// TwinCAT 3 PLC project Oefeningen4
// ProgramVersion: 3.1.4026.18
// libraries:
//   Tc2_BABasic, * (Beckhoff Automation GmbH)
//   Tc2_Standard, * (Beckhoff Automation GmbH)
//   Tc2_System, * (Beckhoff Automation GmbH)
//   Tc2_Utilities, * (Beckhoff Automation GmbH)
//   Tc3_Module, * (Beckhoff Automation GmbH)
// project tree:
//   DUTs/ DUT_Kamer.TcDUT
//   / GlobalTextList.TcGTLO, PlcTask.TcTTO, Visualization Manager.TcVMO (not stored)
//   POUs/ MAIN.TcPOU, MEAN.TcPOU, prg_Finale.TcPOU, prg_KantoorVerlichting.TcPOU, prg_Thermostaatregeling.TcPOU, prg_ThermostaatregelingTijdsturing.TcPOU
//   VISUs/ Visualization_Thermostaatregeling.TcVIS, Visualization_ThermostaatTijdsturing.TcVIS
// (motion and I/O tree: see PLC project oefeningen1)
// real-time tasks:
//   TASK PlcTask: cycle T#10ms, priority 20, ADS port 350
//   TASK PlcTask1: cycle T#10ms, priority 21, ADS port 351
//   TASK PlcTask2: cycle T#10ms, priority 22, ADS port 352
//   TASK PlcTask3: cycle T#10ms, priority 23, ADS port 353
//   TASK PlcTask4: cycle T#10ms, priority 24, ADS port 354

CONFIGURATION Oefeningen4
    RESOURCE PLC ON TwinCAT3
        TASK PlcTask(INTERVAL := T#10ms, PRIORITY := 23);
        PROGRAM MAIN WITH PlcTask : MAIN;
    END_RESOURCE
END_CONFIGURATION

// ---- DUTs/DUT_Kamer.TcDUT
TYPE DUT_Kamer :
STRUCT
    Licht : BOOL;
    Temperatuur : REAL;
    MA_Temp : REAL;
END_STRUCT
END_TYPE

// ---- POUs/MAIN.TcPOU
PROGRAM MAIN
VAR
END_VAR

//prg_KantoorVerlichting();
//prg_Thermostaatregeling();
prg_ThermostaatregelingTijdsturing();

END_PROGRAM

// ---- POUs/prg_ThermostaatregelingTijdsturing.TcPOU
PROGRAM prg_ThermostaatregelingTijdsturing
VAR
   	Temperatuur : REAL;            
    TempLog     : ARRAY[0..19] OF REAL;
    TempAlarm   : ARRAY[0..19] OF BOOL;
    idx         : INT := 0;        
    tSample     : TON;
END_VAR

// timer 1 seconde
tSample(IN := TRUE, PT := T#1S);
tSample();

IF tSample.Q THEN
    TempLog[idx] := Temperatuur;               // log huidige temperatuur
    TempAlarm[idx] := (Temperatuur < 10.0);   // alarm als <10°C
    idx := (idx + 1) MOD 20;                  // circular buffer
    tSample(IN := FALSE);
    tSample(IN := TRUE);
END_IF

END_PROGRAM

// ---- POUs/MEAN.TcPOU
FUNCTION MEAN : REAL
VAR_INPUT
    arr : ARRAY[1..10] OF REAL;
END_VAR

VAR
    i : INT;
    sum : REAL := 0.0;
END_VAR

FOR i := 1 TO 10 DO
    sum := sum + arr[i];
END_FOR

MEAN := sum / 10.0;

END_FUNCTION

// ---- POUs/prg_Finale.TcPOU
PROGRAM prg_Finale
VAR
    (* ---- Kamers ---- *)
    Woonkamer : DUT_Kamer := (Temperatuur := 21.0);
    Keuken    : DUT_Kamer := (Temperatuur := 20.5);
    Badkamer  : DUT_Kamer := (Temperatuur := 22.0);
    Gang      : DUT_Kamer := (Temperatuur := 19.5);

    (* ---- 10s timer ---- *)
    tMeasure : TON;

    (* ---- Moving Average buffers (10 waarden) ---- *)
    TempBuf_WK : ARRAY[1..10] OF REAL;
    TempBuf_K  : ARRAY[1..10] OF REAL;
    TempBuf_B  : ARRAY[1..10] OF REAL;
    TempBuf_G  : ARRAY[1..10] OF REAL;

    idx : INT := 1; (* circulaire index 1..10 *)

    (* ---- Logging MA + timestamp (laatste 20 waarden) ---- *)
    LogMA : ARRAY[1..20, 1..2] OF LREAL;
    (* Kolom 1 = timestamp (s), Kolom 2 = MA temperatuur *)

    logIndex : INT := 1;

    sysTime : LTIME;

    (* ---- VISU toggles ---- *)
    VISU_Toggle_WK : BOOL;
    VISU_Toggle_K  : BOOL;
    VISU_Toggle_B  : BOOL;
    VISU_Toggle_G  : BOOL;

    VISU_ShowTemp : BOOL;
END_VAR

(* Start 10s timer *)
tMeasure(IN := TRUE, PT := T#10s);

(* ---- Licht toggles (via visualisatie) ---- *)
IF VISU_Toggle_WK THEN
    Woonkamer.Licht := NOT Woonkamer.Licht;
    VISU_Toggle_WK := FALSE;
END_IF

IF VISU_Toggle_K THEN
    Keuken.Licht := NOT Keuken.Licht;
    VISU_Toggle_K := FALSE;
END_IF

IF VISU_Toggle_B THEN
    Badkamer.Licht := NOT Badkamer.Licht;
    VISU_Toggle_B := FALSE;
END_IF

IF VISU_Toggle_G THEN
    Gang.Licht := NOT Gang.Licht;
    VISU_Toggle_G := FALSE;
END_IF

(* ---- Elke 10 seconden meten ---- *)
IF tMeasure.Q THEN

    (* Simuleer temperatuur (later vervang je dit door echte sensor) *)
    Woonkamer.Temperatuur := Woonkamer.Temperatuur + (RAND() - 0.5) * 0.2;
    Keuken.Temperatuur    := Keuken.Temperatuur + (RAND() - 0.5) * 0.2;
    Badkamer.Temperatuur  := Badkamer.Temperatuur + (RAND() - 0.5) * 0.2;
    Gang.Temperatuur      := Gang.Temperatuur + (RAND() - 0.5) * 0.2;

    (* ---- Circulaire buffer update ---- *)
    idx := idx + 1;
    IF idx > 10 THEN
        idx := 1;
    END_IF

    TempBuf_WK[idx] := Woonkamer.Temperatuur;
    TempBuf_K[idx]  := Keuken.Temperatuur;
    TempBuf_B[idx]  := Badkamer.Temperatuur;
    TempBuf_G[idx]  := Gang.Temperatuur;

    (* ---- Bereken Moving Average ---- *)
    Woonkamer.MA_Temp := MEAN(TempBuf_WK);
    Keuken.MA_Temp    := MEAN(TempBuf_K);
    Badkamer.MA_Temp  := MEAN(TempBuf_B);
    Gang.MA_Temp      := MEAN(TempBuf_G);

    (* ---- Timestamp ---- *)
    sysTime := F_GetCurTime();

    (* ---- Log laatste 20 MA waarden (voor tabel in VISU) ---- *)
    LogMA[logIndex,1] := LTIME_TO_LREAL(sysTime) / 1_000_000_000.0; (* seconden *)
    LogMA[logIndex,2] := Woonkamer.MA_Temp; (* je kan hier ook andere kamer kiezen *)

    logIndex := logIndex + 1;
    IF logIndex > 20 THEN
        logIndex := 1;
    END_IF

    (* Reset timer *)
    tMeasure(IN := FALSE);
END_IF

END_PROGRAM

// ---- POUs/prg_KantoorVerlichting.TcPOU
PROGRAM prg_KantoorVerlichting
VAR
	bSchakelaar_1		AT		%I*		:BOOL;
	bSchakelaar_2		AT		%I*		:BOOL;
	bSchakelaar_3		AT		%I*		:BOOL;
	bVerlichting	 	AT 		%Q* 	:BOOL;

	LichtVerlengen: TON;
	TimerVerlichting: TP;
	Flikkeraan: TON;
	FlikkerUit: TOF;
	Flikker: REAL;
	Uitklik: F_TRIG;
	bVerlichtingRaw: BOOL;
END_VAR

LichtVerlengen(IN:= bSchakelaar_1, PT:= T#2S);
TimerVerlichting(IN:= bSchakelaar_1 OR LichtVerlengen.Q, PT:= T#60S, Q=> bVerlichting);

IF TIME_TO_REAL(TimerVerlichting.ET) >= 30 AND Flikker < 3 THEN
	Flikkeraan(IN:= NOT(FlikkerUit.Q) , PT:= T#500MS, Q=> bVerlichting);
	FlikkerUit(IN:= Flikkeraan.Q, PT:= T#500MS);
	Flikker := Flikker+1;
END_IF

IF FlikkerUit.Q THEN
	bVerlichting:=NOT(TimerVerlichting.Q);
ELSE
	bVerlichting:=TimerVerlichting.Q;
END_IF

Uitklik(CLK:= bSchakelaar_1);

IF TIME_TO_REAL(TimerVerlichting.ET) >= 30 AND LichtVerlengen.Q THEN
	TimerVerlichting.IN:=TRUE;
ELSIF bVerlichting AND Uitklik.Q AND NOT(LichtVerlengen.Q) THEN
	bVerlichting:=FALSE;
	TimerVerlichting.IN:=FALSE;
END_IF

END_PROGRAM

// ---- POUs/prg_Thermostaatregeling.TcPOU
PROGRAM prg_Thermostaatregeling
VAR
	Thermostaat			AT		%I*		:REAL;
	Potentiometer1		AT		%I*		:INT;
	Potentiometer2		AT		%I*		:INT;
	
	Temperatuur			AT		%Q*		:REAL;
	Verwarming			AT		%Q*		:BOOL; //Is een Lamp
	TijdsRegeling: FB_WeeklyTimeSwitch;
	Dag: BOOL;

    fbTime : FB_LocalSystemTime;
    currentDT : DATE_AND_TIME;
END_VAR

//JE MOET VANONDER DE TIJDEN VAN EN TOT WANNEER AANPASSEN ALS JE DIT PROGRAMMA NIET TUSSEN
// 8u30 en 18u00 test

//SYSTEEM TIJD EN DATUM VOOR DE TIJDSREGELING HIERONDER:
fbTime(bEnable := TRUE);              // één keer starten, daarna cyclisch laten lopen
currentDT := SYSTEMTIME_TO_DT(fbTime.systemTime);

//programma met echte potentiometers van 0-32767:
//Thermostaat := 10.0 + (INT_TO_REAL(Potentiometer1) * 20.0 / 32767.0);
//Temperatuur := -30.0 + (INT_TO_REAL(Potentiometer2) * 70.0 / 32767.0);

//IF (Temperatuur < (Thermostaat - 1.0)) AND Dag THEN
//	Verwarming:=TRUE;
//ELSIF (Temperatuur >= (Thermostaat + 1.0)) OR NOT(Dag) THEN
//	Verwarming:=FALSE;
//END_IF

//Programma met de potentiometers in de visualisatie (anders verschaald)
Thermostaat := Potentiometer1;  // waarde van 10..30°C uit de Visu
Temperatuur := Potentiometer2;  // waarde van -30..40°C uit de Visu

IF (Temperatuur < (Thermostaat - 1.0)) AND Dag THEN
    Verwarming := TRUE;
ELSIF (Temperatuur >= (Thermostaat + 1.0)) OR NOT(Dag) THEN
    Verwarming := FALSE;
END_IF

//FunctieBlok uit library om tijdsinstellingen van 
TijdsRegeling(
	bEnable:= TRUE, 
	tCurrentDateTime:= currentDT, //hier moet een systeem variabele zoals CURRENT_DT of SYSTEM_DATE_AND_TIME maar vind ik niet
	tSwitchOnTime:= TOD#08:30, 
	tSwitchOffTime:= TOD#18:00, 
	bSunday:= TRUE, 
	bMonday:= TRUE, 
	bTuesday:= TRUE, 
	bWednesday:= TRUE, 	
	bThursday:= TRUE, 
	bFriday:= TRUE, 
	bSaturday:= TRUE, 
	bOutput=> Dag);

END_PROGRAM

// ---- GlobalTextList.TcGTLO
TEXTLIST GlobalTextList
  134 = 'Potentioemter2'
  385 = 'Potentiometer1'
  583 = 'Potentiometer2'
  204 = 'Temperatu ur (-30°C - 40°C)'
  232 = 'Temperatuur'
  546 = 'Temperatuur (-30°C - 40°C)'
  8 = 'Thermostaat'
  611 = 'Thermostaat (10°C - 30°C'
  970 = 'Thermostaat (10°C - 30°C)'
END_TEXTLIST

// ---- VISUs/Visualization_Thermostaatregeling.TcVIS
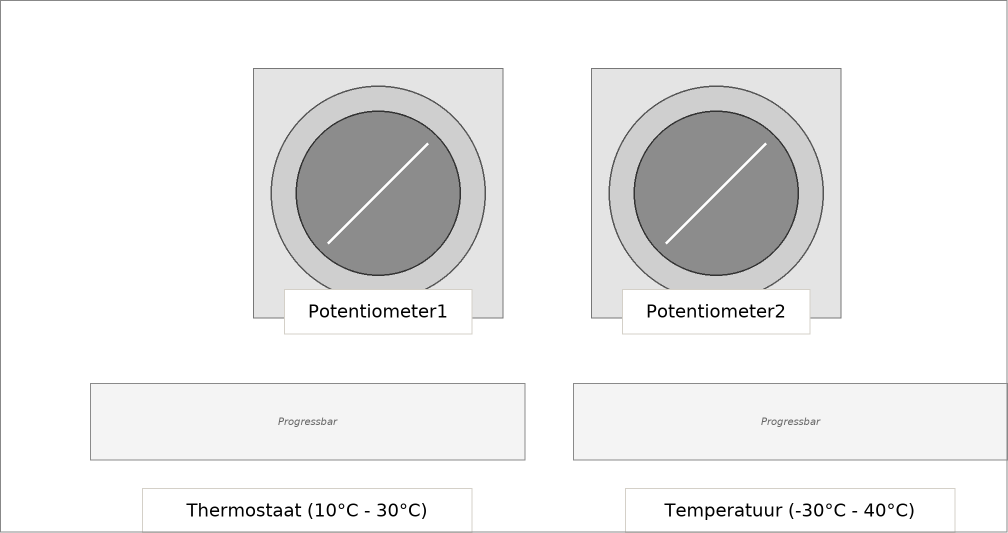
VISUALIZATION Visualization_Thermostaatregeling  // 1008x533
    Potentiometer360 (253,68 250x250), variable: prg_Thermostaatregeling.Potentiometer1, style: Potentiometer-Potentiometer360-Gray, scale format: %.1f, scale 10..30
        p2431819421: Outside
    Potentiometer360 (591,68 250x250), variable: prg_Thermostaatregeling.Potentiometer2, style: Potentiometer-Potentiometer360-Gray, scale format: %.1f, scale -30..40
        p2431819421: Outside
    Textfield (284,289 188x45), "Potentiometer1"
    Textfield (622,289 188x45), "Potentiometer2"
    Progressbar (573,383 435x77), variable: prg_Thermostaatregeling.Temperatuur
    Textfield (625,488 330x45), "Temperatuur (-30°C - 40°C)"
    Progressbar (90,383 435x77), variable: prg_Thermostaatregeling.Thermostaat
    Textfield (142,488 330x45), "Thermostaat (10°C - 30°C)"
END_VISUALIZATION

// ---- VISUs/Visualization_ThermostaatTijdsturing.TcVIS
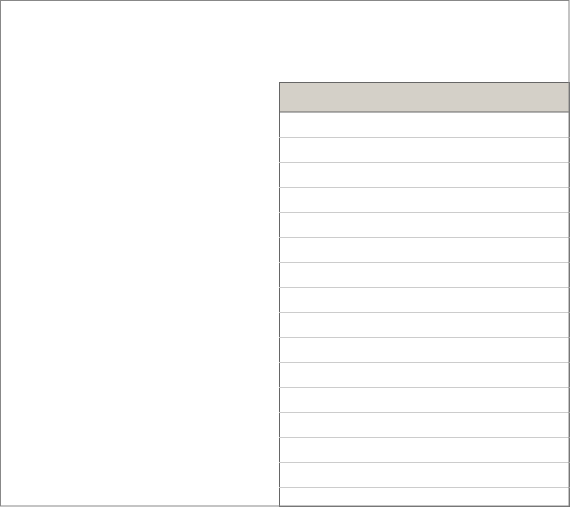
VISUALIZATION Visualization_ThermostaatTijdsturing  // 570x507
    Table (279,82 291x425), data array: prg_ThermostaatregelingTijdsturing.TempLog
        p3854506369: prg_ThermostaatregelingTijdsturing.TempLog[INDEX]
        p2232123230: Temperatuur
        Columns.Column.[0].Template: prg_ThermostaatregelingTijdsturing.TempAlarm
END_VISUALIZATION
